// TIA Portal V15.1 export
// export: Created 2024-06-21T08:40:49.0888547Z, ExportSetting WithDefaults, DisplayName Totally Integrated Automation Portal, DisplayVersion V15.1 Update 5, DisplayName TIA Portal Openness, DisplayVersion V15.1 Update 5, DisplayName SINAMICS Startdrive Advanced, DisplayVersion V15.1, DisplayName G130, G150, S120, S150, SINAMICS MV, S210, DisplayVersion V15.1, DisplayName G110M, G120, G120C, G120D, G120P, DisplayVersion V15.1, DisplayName STEP 7 Professional, DisplayVersion V15.1 Update 5, DisplayName STEP 7 Safety, DisplayVersion V15.1, DisplayName WinCC Professional, DisplayVersion V15.1 Update 5, DisplayName SIMATIC Visualization Architect, DisplayVersion V15.1
DATA_BLOCK "_209220ZM01DataHandling"   // DB354
{ S7_Optimized_Access := 'FALSE' }
AUTHOR : VCC
VERSION : 0.1
// stored: AutoNumber false, DBAccessibleFromOPCUA true, IsOnlyStoredInLoadMemory false, IsWriteProtectedInAS false
   VAR RETAIN
      AC_209220NCB01VIDSMasterAlarm { ExternalAccessible := 'False'; ExternalVisible := 'False'; ExternalWritable := 'False'} : Bool;   // VIDS 209220NCB01 - Master Alarm
      AC_209220NCB01VIDSRFIDAlarm { ExternalAccessible := 'False'; ExternalVisible := 'False'; ExternalWritable := 'False'} : Bool;   // VIDS 209220NCB01 - RFID Alarm
      AC_209220NCB01VIDSTrackingAlarm { ExternalAccessible := 'False'; ExternalVisible := 'False'; ExternalWritable := 'False'} : Bool;   // VIDS 209220NCB01 - Tracking Alarm
      AC_209220NCB02VIDSMasterAlarm { ExternalAccessible := 'False'; ExternalVisible := 'False'; ExternalWritable := 'False'} : Bool;   // VIDS 209220NCB02 - Master Alarm
      AC_209220NCB02VIDSRFIDAlarm { ExternalAccessible := 'False'; ExternalVisible := 'False'; ExternalWritable := 'False'} : Bool;   // VIDS 209220NCB02 - RFID Alarm
      AC_209220NCB02VIDSQualityRequestAlarm { ExternalAccessible := 'False'; ExternalVisible := 'False'; ExternalWritable := 'False'} : Bool;   // VIDS 209220NCB02 - Quality Request Alarm
      AC_209220NCB02VIDSTrackingAlarm { ExternalAccessible := 'False'; ExternalVisible := 'False'; ExternalWritable := 'False'} : Bool;   // VIDS 209220NCB02 - Tracking Alarm
      H_HMICmd : Word;   // Commands from HMI
      H_Anim : Word;   // Animation
      H_DBnr : Int;   // DB number
      H_209220NCB01TagSequenceIAnim : Word;   // Icon Animation
      H_209220NCB02TagSequenceIAnim : Word;   // Icon Animation
      H_HMI : Struct   // HMI Animation
         "209220NCB01VIDSMaster" : "H_HMI";   // HMI Animation
         "209220NCB01VIDSRFID" : "H_HMI";   // HMI Animation
         "209220NCB01VIDSTracking" : "H_HMI";   // HMI Animation
         "209220NCB02VIDSMaster" : "H_HMI";   // HMI Animation
         "209220NCB02VIDSRFID" : "H_HMI";   // HMI Animation
         "209220NCB02VIDSQualityRequest" : "H_HMI";   // HMI Animation
         "209220NCB02VIDSTracking" : "H_HMI";   // HMI Animation
      END_STRUCT;
      H : Struct   // HMI Animation
         "209220NCB01VIDSMaster" : "H_LVIDSMaster";   // HMI Animation
         "209220NCB01VIDSRFID" : "H_LVIDSRFID";   // HMI Animation
         "209220NCB01VIDSTracking" : "H_LVIDSTrack";   // HMI Animation
         "209220NCB02VIDSMaster" : "H_LVIDSMaster";   // HMI Animation
         "209220NCB02VIDSRFID" : "H_LVIDSRFID";   // HMI Animation
         "209220NCB02VIDSQualityRequest" : "H_LVIDSQualityRequest";   // HMI Animation
         "209220NCB02VIDSTracking" : "H_LVIDSTrack";   // HMI Animation
      END_STRUCT;
      AlarmABCondition { ExternalAccessible := 'False'; ExternalVisible := 'False'; ExternalWritable := 'False'} : Bool;   // Alarm AB condition
      AlarmA { ExternalAccessible := 'False'; ExternalVisible := 'False'; ExternalWritable := 'False'} : Bool;   // Alarm A
      AlarmB { ExternalAccessible := 'False'; ExternalVisible := 'False'; ExternalWritable := 'False'} : Bool;   // Alarm B
      AlarmC { ExternalAccessible := 'False'; ExternalVisible := 'False'; ExternalWritable := 'False'} : Bool;   // Alarm C
      AlarmD { ExternalAccessible := 'False'; ExternalVisible := 'False'; ExternalWritable := 'False'} : Bool;   // Alarm D
      "209220NCB01TagSequence" { ExternalAccessible := 'False'; ExternalVisible := 'False'; ExternalWritable := 'False'} : "AlarmBits";   // Tag Sequence Alarm Bits
      "209220NCB01ReadBegin" { ExternalAccessible := 'False'; ExternalVisible := 'False'; ExternalWritable := 'False'} : Bool;   // Start Reading Body Data
      "209220NCB01BodyData" { ExternalAccessible := 'False'; ExternalVisible := 'False'; ExternalWritable := 'False'; S7_SetPoint := 'True'} : "VEMData";   // Body Data from VEMData
      "209220NCB02TagSequence" { ExternalAccessible := 'False'; ExternalVisible := 'False'; ExternalWritable := 'False'} : "AlarmBits";   // Tag Sequence Alarm Bits
      "209220NCB02ReadBegin" { ExternalAccessible := 'False'; ExternalVisible := 'False'; ExternalWritable := 'False'} : Bool;   // Start Reading Body Data
      "209220NCB02BodyData" { ExternalAccessible := 'False'; ExternalVisible := 'False'; ExternalWritable := 'False'; S7_SetPoint := 'True'} : "VEMData";   // Body Data from VEMData
      "______209220NCB01_VIDS Master______" { ExternalAccessible := 'False'; ExternalVisible := 'False'; ExternalWritable := 'False'} : Bool;   // -----------------------------------------------------------------------------------
      "209220NCB01VIDS" { ExternalAccessible := 'False'; ExternalVisible := 'False'; ExternalWritable := 'False'; S7_SetPoint := 'True'} : "VIDS";   // Internal record
      "209220NCB01VEMData" { ExternalAccessible := 'False'; ExternalVisible := 'False'; ExternalWritable := 'False'; S7_SetPoint := 'True'} : "VEMData";   // VEM Data
      "209220NCB01VEMDataChange" { ExternalAccessible := 'False'; ExternalVisible := 'False'; ExternalWritable := 'False'; S7_SetPoint := 'True'} : "VEMData";   // VEM Data Change
      "209220NCB01VEMDataValid" { ExternalAccessible := 'False'; ExternalVisible := 'False'; ExternalWritable := 'False'; S7_SetPoint := 'True'} : Bool;   // VEM Data Valid
      "209220NCB01VEMDataNotValid" { ExternalAccessible := 'False'; ExternalVisible := 'False'; ExternalWritable := 'False'; S7_SetPoint := 'True'} : Bool;   // VEM Data Not Valid
      "209220NCB01GetVEMDataBusy" { ExternalAccessible := 'False'; ExternalVisible := 'False'; ExternalWritable := 'False'; S7_SetPoint := 'True'} : Bool;   // Get VEM Data Busy
      "209220NCB01MasterStatus" { ExternalAccessible := 'False'; ExternalVisible := 'False'; ExternalWritable := 'False'; S7_SetPoint := 'True'} : Int;   // Master - Status
      "______209220NCB01_VIDS RFID______" { ExternalAccessible := 'False'; ExternalVisible := 'False'; ExternalWritable := 'False'} : Bool;   // -----------------------------------------------------------------------------------
      "209220NCB01ReadOK" { ExternalAccessible := 'False'; ExternalVisible := 'False'; ExternalWritable := 'False'; S7_SetPoint := 'True'} : Bool;   // RFID - Read OK
      "209220NCB01ReadNOK" { ExternalAccessible := 'False'; ExternalVisible := 'False'; ExternalWritable := 'False'; S7_SetPoint := 'True'} : Bool;   // RFID - Read NOK
      "209220NCB01Busy" { ExternalAccessible := 'False'; ExternalVisible := 'False'; ExternalWritable := 'False'; S7_SetPoint := 'True'} : Bool;   // RFID - Busy
      "209220NCB01Status" { ExternalAccessible := 'False'; ExternalVisible := 'False'; ExternalWritable := 'False'; S7_SetPoint := 'True'} : Int;   // RFID - Status
      "______209220NCB01_VIDS Tracking______" { ExternalAccessible := 'False'; ExternalVisible := 'False'; ExternalWritable := 'False'} : Bool;   // -----------------------------------------------------------------------------------
      "209220NCB01TrackOK" { ExternalAccessible := 'False'; ExternalVisible := 'False'; ExternalWritable := 'False'; S7_SetPoint := 'True'} : Bool;   // Track - OK
      "209220NCB01TrackNOK" { ExternalAccessible := 'False'; ExternalVisible := 'False'; ExternalWritable := 'False'; S7_SetPoint := 'True'} : Bool;   // Track - Nok
      "209220NCB01TrackBusy" { ExternalAccessible := 'False'; ExternalVisible := 'False'; ExternalWritable := 'False'; S7_SetPoint := 'True'} : Bool;   // Track - Busy
      "209220NCB01TrackStatus" { ExternalAccessible := 'False'; ExternalVisible := 'False'; ExternalWritable := 'False'; S7_SetPoint := 'True'} : Int;   // Track - Status
      "209220NCB01SpecificData" { ExternalAccessible := 'False'; ExternalVisible := 'False'; ExternalWritable := 'False'; S7_SetPoint := 'True'} : Array[0..7925] of Byte;   // Specific Data Received
      "______209220NCB02_VIDS Master______" { ExternalAccessible := 'False'; ExternalVisible := 'False'; ExternalWritable := 'False'} : Bool;   // -----------------------------------------------------------------------------------
      "209220NCB02VIDS" { ExternalAccessible := 'False'; ExternalVisible := 'False'; ExternalWritable := 'False'; S7_SetPoint := 'True'} : "VIDS";   // Internal record
      "209220NCB02VEMData" { ExternalAccessible := 'False'; ExternalVisible := 'False'; ExternalWritable := 'False'; S7_SetPoint := 'True'} : "VEMData";   // VEM Data
      "209220NCB02VEMDataChange" { ExternalAccessible := 'False'; ExternalVisible := 'False'; ExternalWritable := 'False'; S7_SetPoint := 'True'} : "VEMData";   // VEM Data Change
      "209220NCB02VEMDataValid" { ExternalAccessible := 'False'; ExternalVisible := 'False'; ExternalWritable := 'False'; S7_SetPoint := 'True'} : Bool;   // VEM Data Valid
      "209220NCB02VEMDataNotValid" { ExternalAccessible := 'False'; ExternalVisible := 'False'; ExternalWritable := 'False'; S7_SetPoint := 'True'} : Bool;   // VEM Data Not Valid
      "209220NCB02GetVEMDataBusy" { ExternalAccessible := 'False'; ExternalVisible := 'False'; ExternalWritable := 'False'; S7_SetPoint := 'True'} : Bool;   // Get VEM Data Busy
      "209220NCB02MasterStatus" { ExternalAccessible := 'False'; ExternalVisible := 'False'; ExternalWritable := 'False'; S7_SetPoint := 'True'} : Int;   // Master - Status
      "______209220NCB02_VIDS RFID______" { ExternalAccessible := 'False'; ExternalVisible := 'False'; ExternalWritable := 'False'} : Bool;   // -----------------------------------------------------------------------------------
      "209220NCB02ReadOK" { ExternalAccessible := 'False'; ExternalVisible := 'False'; ExternalWritable := 'False'; S7_SetPoint := 'True'} : Bool;   // RFID - Read OK
      "209220NCB02ReadNOK" { ExternalAccessible := 'False'; ExternalVisible := 'False'; ExternalWritable := 'False'; S7_SetPoint := 'True'} : Bool;   // RFID - Read NOK
      "209220NCB02Busy" { ExternalAccessible := 'False'; ExternalVisible := 'False'; ExternalWritable := 'False'; S7_SetPoint := 'True'} : Bool;   // RFID - Busy
      "209220NCB02Status" { ExternalAccessible := 'False'; ExternalVisible := 'False'; ExternalWritable := 'False'; S7_SetPoint := 'True'} : Int;   // RFID - Status
      "______209220NCB02_VIDS Quality Request______" { ExternalAccessible := 'False'; ExternalVisible := 'False'; ExternalWritable := 'False'} : Bool;   // -----------------------------------------------------------------------------------
      "209220NCB02Quality RequestDataValid" { ExternalAccessible := 'False'; ExternalVisible := 'False'; ExternalWritable := 'False'; S7_SetPoint := 'True'} : Bool;   // Quality Request - Data Valid
      "209220NCB02Quality RequestDataNotValid" { ExternalAccessible := 'False'; ExternalVisible := 'False'; ExternalWritable := 'False'; S7_SetPoint := 'True'} : Bool;   // Quality Request - Data Not Valid
      "209220NCB02Quality RequestBusy" { ExternalAccessible := 'False'; ExternalVisible := 'False'; ExternalWritable := 'False'; S7_SetPoint := 'True'} : Bool;   // Quality Request - Busy
      "209220NCB02Quality RequestStatus" { ExternalAccessible := 'False'; ExternalVisible := 'False'; ExternalWritable := 'False'; S7_SetPoint := 'True'} : Int;   // Quality Request - Status
      "209220NCB02Quality RequestVEMData" { ExternalAccessible := 'False'; ExternalVisible := 'False'; ExternalWritable := 'False'; S7_SetPoint := 'True'} : "VEMData";   // Quality Request - VEM Data
      "______209220NCB02_VIDS Tracking______" { ExternalAccessible := 'False'; ExternalVisible := 'False'; ExternalWritable := 'False'} : Bool;   // -----------------------------------------------------------------------------------
      "209220NCB02TrackOK" { ExternalAccessible := 'False'; ExternalVisible := 'False'; ExternalWritable := 'False'; S7_SetPoint := 'True'} : Bool;   // Track - OK
      "209220NCB02TrackNOK" { ExternalAccessible := 'False'; ExternalVisible := 'False'; ExternalWritable := 'False'; S7_SetPoint := 'True'} : Bool;   // Track - Nok
      "209220NCB02TrackBusy" { ExternalAccessible := 'False'; ExternalVisible := 'False'; ExternalWritable := 'False'; S7_SetPoint := 'True'} : Bool;   // Track - Busy
      "209220NCB02TrackStatus" { ExternalAccessible := 'False'; ExternalVisible := 'False'; ExternalWritable := 'False'; S7_SetPoint := 'True'} : Int;   // Track - Status
      "209220NCB02SpecificData" { ExternalAccessible := 'False'; ExternalVisible := 'False'; ExternalWritable := 'False'; S7_SetPoint := 'True'} : Array[0..7925] of Byte;   // Specific Data Received
   END_VAR
BEGIN
END_DATA_BLOCK
